Yaskawa INFORM job: R1_W43-44-A1(80,0))KM-OK.JBI

/JOB
//NAME R1_W43-44-A1(80,0))KM-OK
///FOLDERNAME KRIS-SCIANA
//POS
///NPOS 73,73,0,2,0,0
///TOOL 0
///POSTYPE PULSE
///PULSE
C00000=39340,-156269,-131125,-10811,20628,87799
C00001=94745,-160008,-130129,-2582,7638,63771
C00002=96654,-34778,-71054,-19792,73704,55692
C00003=94277,-33017,-66948,-18725,71664,55228
C00004=93802,-33152,-64581,-18638,70115,55316
C00005=93546,-32956,-64450,-18503,70082,55233
C00006=93963,-32178,-66338,-18557,71651,55125
C00007=85606,-7402,-55752,-6638,82644,57380
C00008=85920,-6491,-54240,-6787,82209,57497
C00009=95227,-3822,-50082,-23095,84917,56051
C00010=79791,-31574,-66926,2477,69314,50449
C00011=79730,-32028,-66762,2516,68982,50421
C00012=86027,-43246,-68268,-8769,57741,51016
C00013=86808,-44938,-70357,-9267,58234,51267
C00014=88852,-49125,-75499,-10553,59467,51911
C00015=100000,206,-63012,-22880,98600,38374
C00016=103669,4873,-66726,-33667,97255,62125
C00017=98217,-20490,-79916,-26548,76072,68092
C00018=97507,-20705,-77735,-26273,74586,68220
C00019=98229,-21086,-77900,-26719,74682,68416
C00020=98659,-21058,-77645,-26993,74667,68552
C00021=98798,-21324,-77280,-27118,74378,68663
C00022=100677,-19799,-82098,-27857,78205,68311
C00023=71270,4147,-82602,17131,105074,40619
C00024=68705,2720,-75332,18566,100647,38866
C00025=101326,5644,-66066,-32582,96592,61641
C00026=100352,7901,-65558,-32199,97047,61232
C00027=68705,2720,-75332,18566,100647,38866
C00028=86151,5323,-73272,-7381,99951,48427
C00029=89957,7110,-71038,-13385,100137,50467
C00030=99237,14312,-61052,-28253,99416,54591
C00031=90965,9004,-76328,-15492,99256,51022
C00032=94335,-7981,-65632,-23039,101372,-9650
C00033=82460,11976,-50910,-8916,109868,-9457
C00034=81792,11917,-50588,-8743,109585,-9630
C00035=103096,-21273,-76552,-41945,77376,-71035
C00036=103793,-24634,-77705,-42464,76882,-70571
C00037=69550,16972,-45708,6116,108518,-27115
C00038=63907,33649,-28963,16122,112033,-40802
C00039=65630,38063,-23798,15706,110881,-40423
C00040=65273,39151,-22632,15751,110787,-40547
C00041=63636,54279,-5451,20327,115064,-51969
C00042=61254,50960,-6170,22648,115588,-46011
C00043=63719,40856,-22586,16130,111852,-40883
C00044=62886,41129,-23270,16352,112524,-41049
C00045=43952,29149,-14118,46602,107199,-63920
C00046=43952,29149,-14118,46602,107199,-63920
C00047=44842,27780,-15084,46451,106700,-63753
C00048=43924,28854,-13411,46455,106801,-64132
C00049=43913,26730,-16470,46663,107362,-63858
C00050=44380,26112,-14250,46173,105957,-64334
C00051=43958,28522,-13185,46372,106567,-64232
C00052=42943,33668,-10503,46768,107748,-64117
C00053=50946,14174,-44109,28846,101382,-67604
C00054=65589,2823,-51194,13094,89139,-67789
C00055=66656,5544,-48857,12654,88957,-67500
C00056=58397,20795,-36993,26400,98477,-65921
C00057=63589,9335,-47554,24733,97708,-64463
C00058=64233,7735,-47405,24457,96714,-64474
C00059=64924,9391,-45783,24215,96406,-64321
C00060=63898,11525,-49886,24841,99966,-63891
C00061=66059,-18193,-73083,5807,84664,-70915
C00062=70495,-21842,-63875,3692,76925,-69924
C00063=76118,-30577,-70021,865,76077,-68221
C00064=74993,-27941,-76004,1411,81127,-68508
C00065=71632,-2103,-60605,3063,85004,-69381
C00066=68491,-10706,-57969,10689,77137,-68380
C00067=75161,-21469,-65891,7214,75849,-66461
C00068=73728,-23153,-69742,7928,77455,-66791
C00069=66211,-30081,-97440,11666,91458,-67720
C00070=94360,-29213,-96879,11541,91532,-67653
C00071=94745,-160008,-130129,-2582,7638,63771
C00072=19116,-160008,-130129,-2582,7638,63771
BC00000=182726,733572,1062903
BC00001=1250,1191141,1062776
BC00002=1194,1191142,1062845
BC00003=1194,1191142,1062845
BC00004=1194,1191142,1062845
BC00005=1194,1191142,1062845
BC00006=1194,1191142,1062845
BC00007=1194,1191142,1062845
BC00008=1194,1191142,1062845
BC00009=1194,1191142,1062845
BC00010=1194,1191142,1062845
BC00011=1194,1191142,1062845
BC00012=1194,1191142,1062845
BC00013=1194,1191142,1062845
BC00014=1194,1191142,1062845
BC00015=1194,1191142,994179
BC00016=1194,1191142,915703
BC00017=1194,1191142,886057
BC00018=1194,1191142,886057
BC00019=1194,1191142,886057
BC00020=1194,1191142,886057
BC00021=1194,1191142,886057
BC00022=1194,1191142,886057
BC00023=1194,1191142,886057
BC00024=1194,1191142,886057
BC00025=1194,1191142,888813
BC00026=1194,1191142,888813
BC00027=1194,1191142,886057
BC00028=1194,1191142,886057
BC00029=1194,1191142,886057
BC00030=1194,1191142,886057
BC00031=1194,1191142,886055
BC00032=1194,1191142,1036504
BC00033=1195,1191142,1035519
BC00034=1195,1191142,1035519
BC00035=1194,1191142,889738
BC00036=1194,1191142,889738
BC00037=1195,1191142,1035519
BC00038=1195,1191141,1035516
BC00039=1195,1191141,1035516
BC00040=1195,1191141,1035516
BC00041=1195,1191141,1035516
BC00042=1195,1191141,1035516
BC00043=1195,1191141,1035516
BC00044=1195,1191141,1035516
BC00045=1194,1168747,1062845
BC00046=1194,1168747,1062845
BC00047=1194,1167505,1062845
BC00048=1194,1167505,1062845
BC00049=1194,1167505,1062845
BC00050=1194,1170669,1062845
BC00051=1194,1171910,1062845
BC00052=1194,1175015,1062845
BC00053=1194,1175015,1062845
BC00054=1194,1175015,1062845
BC00055=1194,1175015,1062845
BC00056=1194,1175015,1062845
BC00057=1194,1175015,1062845
BC00058=1194,1175015,1062845
BC00059=1194,1175015,1062845
BC00060=1194,1175015,1062845
BC00061=1194,1175015,1062843
BC00062=1194,1175015,1062843
BC00063=1194,1175015,1062843
BC00064=1194,1175015,1062843
BC00065=1194,1175015,1062843
BC00066=1194,1175015,1062843
BC00067=1194,1175015,1062843
BC00068=1194,1175015,1062843
BC00069=1194,1175015,1062843
BC00070=1194,1175015,1062843
BC00071=1250,1163535,1062776
BC00072=60102,670455,1062776
///POSTYPE BASE
///RECTAN
///RCONF 0,0,0,0,0,0,0,0,0,0,0,0,0,0,0,0,0,0,0,0,0,0,0,0
P00006=0.222,-3.123,-1.508,0.0000,0.0000,0.0000
P00023=0.143,-0.036,0.682,0.0000,0.0000,0.0000
//INST
///DATE 2024/07/24 14:50
///ATTR SC,RW
///GROUP1 RB1,BS1
NOP
'r1_W43-44-A1(80,0))
'Path S1224
MOVJ C00000 BC00000 VJ=100.00
MOVJ C00001 BC00001 VJ=100.00
SFTOF
MOVJ C00002 BC00002 VJ=100.00
MOVJ C00003 BC00003 VJ=100.00
MOVL C00004 BC00004 V=60.0
REFP 3 C00005 BC00005
CALL JOB:SEARCH-R1
SET P023 P006
SFTON P023
MOVL C00006 BC00006 V=60.0
MOVL C00007 BC00007 V=60.0
REFP 3 C00008 BC00008
CALL JOB:SEARCH-R1
SET P023 P006
SFTON P023
MOVL C00009 BC00009 V=60.0
MOVL C00010 BC00010 V=60.0
REFP 3 C00011 BC00011
CALL JOB:SEARCH-R1
SET P023 P006
SFTON P023
MOVL C00012 BC00012 V=60.0
MOVL C00013 BC00013 V=166.7
MOVL C00014 BC00014 V=166.7
'Path VIA1253
SFTOF
MOVJ C00015 BC00015 VJ=100.00
'Path W1225
SFTOF
SFTON P023
MOVJ C00016 BC00016 VJ=100.00
MACRO1 MJ#(0) ARGF7
MOVJ C00017 BC00017 VJ=100.00
MOVJ C00018 BC00018 VJ=100.00
ARCON
MOVL C00019 BC00019 V=8.3
MOVL C00020 BC00020 V=8.3
MOVL C00021 BC00021 V=8.3
ARCOF
MOVJ C00022 BC00022 VJ=15.00
MOVJ C00023 BC00023 VJ=100.00
MOVL C00024 BC00024 V=100.0 PL=0
REFP 1 C00025 BC00025
REFP 2 C00026 BC00026
MACRO1 MJ#(0) ARGF7
ARCON
MOVL C00027 BC00027 V=10.0
MOVL C00028 BC00028 V=10.0
MOVL C00029 BC00029 V=10.0
MOVL C00030 BC00030 V=10.0
ARCOF
MOVL C00031 BC00031 V=166.7
MOVL C00032 BC00032 V=166.7
'Path W1226
SFTOF
SFTON P023
MOVJ C00033 BC00033 VJ=100.00
MOVL C00034 BC00034 V=100.0 PL=0
REFP 1 C00035 BC00035
REFP 2 C00036 BC00036
MACRO1 MJ#(0) ARGF7
ARCON
MOVL C00037 BC00037 V=10.0
MOVL C00038 BC00038 V=10.0
MOVL C00039 BC00039 V=10.0
MACRO1 MJ#(0) ARGF7
MOVL C00040 BC00040 V=8.3
MOVL C00041 BC00041 V=8.3
MOVL C00042 BC00042 V=8.3
ARCOF
MOVL C00043 BC00043 V=166.7
MOVL C00044 BC00044 V=166.7
SFTOF
COMM 'Path VIA1252
COMM SFTON P023
COMM MOVJ C00045 BC00045 VJ=100.00
COMM SFTOF
COMM SFTON P023
COMM MOVJ C00046 BC00046 VJ=100.00
COMM MOVL C00047 BC00047 V=100.0 PL=0
COMM REFP 1 C00048 BC00048
COMM REFP 2 C00049 BC00049
COMM MACRO1 MJ#(0) ARGF9
COMM ARCON
COMM MOVL C00050 BC00050 V=10.0
COMM ARCOF
COMM MOVL C00051 BC00051 V=166.7
COMM MOVL C00052 BC00052 V=166.7
COMM SFTOF
COMM MOVJ C00053 BC00053 VJ=100.00
COMM MACRO1 MJ#(0) ARGF6
COMM MOVJ C00054 BC00054 VJ=100.00
COMM 'ARCON
COMM MOVL C00055 BC00055 V=8.3
COMM 'ARCOFF
COMM MOVJ C00056 BC00056 VJ=100.00
COMM MOVJ C00057 BC00057 VJ=100.00
COMM MOVJ C00058 BC00058 VJ=100.00
COMM 'ARCON
COMM MOVL C00059 BC00059 V=9.2
COMM 'ARCOFF
COMM MOVJ C00060 BC00060 VJ=100.00
MOVJ C00061 BC00061 VJ=100.00
SFTON P023
MOVJ C00062 BC00062 VJ=100.00
ARCON
TIMER T=0.50
ARCOF
MOVJ C00063 BC00063 VJ=100.00
ARCON
TIMER T=0.50
ARCOF
MOVJ C00064 BC00064 VJ=100.00
MOVJ C00065 BC00065 VJ=100.00
MACRO1 MJ#(0) ARGF7
MOVJ C00066 BC00066 VJ=100.00
ARCON
MOVL C00067 BC00067 V=7.5
ARCOF
MOVJ C00068 BC00068 VJ=20.00
SFTOF
MOVJ C00069 BC00069 VJ=100.00
MOVJ C00070 BC00070 VJ=100.00
MOVJ C00071 BC00071 VJ=100.00
MOVJ C00072 BC00072 VJ=100.00
SFTOF
END
